// Convert normalized value to analog value
FUNCTION AnalogOutputConversion : WORD
VAR_INPUT
	ScaledValue : REAL;
END_VAR
VAR
	NormalizedValue : REAL;
END_VAR

VAR_OUTPUT
	AnalogOutput: WORD;
END_VAR

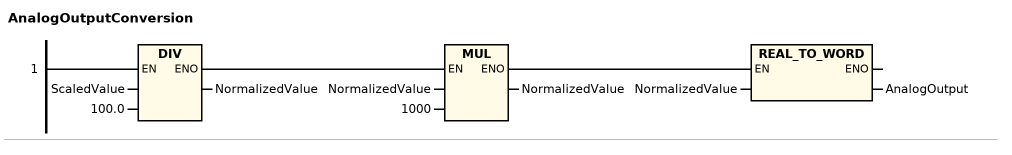
// NETWORK 1
NormalizedValue := ScaledValue / 100.0;
NormalizedValue := NormalizedValue * 1000;
AnalogOutput := REAL_TO_WORD(NormalizedValue);

END_FUNCTION

(* stored: Version 1.1.0.1, ProductVersion 3.1.4024.12
   POU AnalogOutputConversion: Id {ac0c7ab5-d265-4bb5-b5f2-07febe8b25e9}, SpecialFunc None *)
